PROGRAM MAIN
VAR
END_VAR

END_PROGRAM

(* stored: Version 1.1.0.1, ProductVersion 3.1.4024.12
   POU MAIN: Id {3778b533-5767-411e-a006-a9893ad0a5b8}, SpecialFunc None *)
